(*
:Description: Build a W3C traceparent header by hashing domain identifiers
into the trace_id and (optional) parent_span_id positions.

Returns the canonical 55-char string ``00-<trace>-<span>-01`` where:

* ``<trace>`` is ``F_HashTraceId(sTraceId)`` — a 32-hex digest of any
  domain identifier naming the trace (workpiece ID, order ID, session
  ID, …). Every PLC that hashes the same ``sTraceId`` produces the
  same trace_id, so their spans aggregate under one trace in Tempo
  without any explicit traceparent handoff.
* ``<span>`` is ``F_HashSpanId(sParentId)`` when ``sParentId`` is
  non-empty, or 16 zeros when empty. The all-zero form is the
  OTel-defined "no parent" marker; tc-otel treats the consumer span
  as root within its trace.

Typical use: **brownfield aggregation** where MES / DB / barcode gives
you a business identifier (order_id, workpiece_id, batch_id) but not
a pre-minted traceparent. Every station hashing the same sTraceId
aggregates its spans into one Tempo trace.

Example (aggregation-only; sibling spans under one trace_id):

    sTp := F_TraceParentFromString(sTraceId := 'WP-1234');
    spn.Begin(sName := 'station_weigh', sTraceParent := sTp);

Example (explicit chain — consumer cites an upstream producer):

    sTp := F_TraceParentFromString(
        sTraceId  := 'WP-1234',
        sParentId := 'station_weigh');          // name of upstream span
    spn.Begin(sName := 'station_inspect', sTraceParent := sTp);

For true distributed tracing with a transport carrying traceparent
between producers and consumers, prefer forwarding
``PRG_TaskLog.Span.CurrentTraceParent()`` — it returns the exact bytes
tc-otel stored, so multi-hop chains stay consistent without relying
on hash agreement.
*)
FUNCTION F_TraceParentFromString : STRING(60)
VAR_INPUT
    sTraceId  : STRING(80);                 (* identifier hashed via F_HashTraceId → 32-hex trace_id *)
    sParentId : STRING(80) := '';           (* identifier hashed via F_HashSpanId → 16-hex span_id;
                                               empty = no parent (all-zero span_id) *)
END_VAR
VAR
    sTraceHex : STRING(32);
    sSpanHex  : STRING(16);
END_VAR


sTraceHex := F_HashTraceId(sTraceId);

(* Validate sender span_id: must be exactly 16 hex chars, otherwise
   fall back to the all-zero "no parent" marker. This keeps malformed
   callers from producing invalid W3C headers that tc-otel would
   reject. *)
   
IF sParentId <> '' THEN
    sSpanHex := F_HashSpanId(sParentId);
ELSE
    sSpanHex := '0000000000000000';  (* W3C: all-zero span_id = "invalid", signals no parent *)
END_IF

F_TraceParentFromString := CONCAT(
    CONCAT(
        CONCAT('00-', sTraceHex),
        CONCAT('-', sSpanHex)),
    '-01');

END_FUNCTION

(* stored: Version 1.1.0.1, ProductVersion 3.1.4026.18
   POU F_TraceParentFromString: Id {8c9d0e1f-2a3b-4c5d-6e7f-8a9b0c1d2e3f}, SpecialFunc None *)
